// TIA Portal project "ServoPulseHariciPozisyonlama" (V17)

(* hardware
DEVICE "S7-1200 station_1"  S7-1200 Station
   slot 0: "Rack_0"  S7-1200 Rack  Rack  V1.0
   slot 1: "PLC_1"  CPU 1214C DC/DC/DC  6ES7 214-1AG40-0XB0  V4.5
DEVICE "PC-System_1"  SIMATIC PC station
   slot 0: "SIMATIC PC station"  Rail  SIMATIC PC-Station  V1.0
      slot 125: "Stationmanager"  Station_Manager  V6.0.4
   slot 1: "HMI_RT_1"  WinCC RT Advanced  6AV2 104-0xxxx-xxxx  17.0.0.0
      slot 33792: "Computer interface"  Host interface
*)

// ===== PLC "PLC_1"  CPU 1214C DC/DC/DC =====

VAR_GLOBAL   // PLC tag table "Default tag table"
   "Axis_1_Pulse" AT %Q0.0 : Bool;
   "Axis_1_Direction" AT %Q0.1 : Bool;
   "Axis_1_DriveEnable" AT %Q0.2 : Bool;
   "Axis_1_LowHwLimitSwitch" AT %I0.0 : Bool;
   "Axis_1_HighHwLimitSwitch" AT %I0.1 : Bool;
   "SERVO ON/OFF-MC POWER" AT %M0.0 : Bool;
   "Tag_1" AT %M100.0 : Bool;
   "Tag_2" AT %M100.1 : Bool;
   "Tag_3" AT %M100.2 : Bool;
   "Tag_4" AT %MD120 : DWord;
   "Tag_5" AT %MD130 : DWord;
   "Tag_6" AT %MW120 : Word;
   "Tag_7" AT %MW130 : Word;
   "MANUEL İLERİ" AT %M0.1 : Bool;
   "MANUEL GERİ" AT %M0.2 : Bool;
   "MANUEL HIZ DEĞERİ" AT %MD50 : Real;
   "BAŞLANGIÇ NOKTASINA GİT ATA-HOME" AT %M0.3 : Bool;
   "HOME POZİSYON DEĞERİ" AT %MD60 : Real;
   "Tag_10" AT %MB1000 : Byte;
   "HOME MOD DEĞERLERİ" AT %MW1000 : Int;
   "Axis_1_Homing switch" AT %I0.7 : Bool;
   "İSTENEN HEDEFE GİT-ABSOLUTE" AT %M0.4 : Bool;
   "İSTENEN HEDEF-ABSOLUTE" AT %MD100 : Real;
   "HEDEFE GİTME HIZI-ABSOLUTE" AT %MD104 : Real;
   "İSTENEN MESAFE KADAR GİT-RELATİVE" AT %M0.5 : Bool;
   "MESAFE-RELATİVE" AT %MD200 : Real;
   "RELATİVE-HIZ" AT %MD204 : Real;
   "HATA RESET" AT %M0.6 : Bool;
   "RAMPALI DUR-HALT" AT %M0.7 : Bool;
   "MOVE VELOCİTY HIZ ATA" AT %M1.0 : Bool;
   "MOVEVELOCİTY-CURRENT" AT %M1.2 : Bool;
   "PARAMETRE DEĞİŞTİR CHANGEDYNAMİC" AT %M1.3 : Bool;
   "KALKIŞ PARAMETRESİ CHANGE DYNAMİC" AT %M1.4 : Bool;
   "DURMA RAMPASI-CHANGE DYNAMİC" AT %M1.5 : Bool;
   "ACİL STOP DEĞİŞTİR- CHANGE" AT %M1.6 : Bool;
   "YUMUŞATMA ZAMANI DEĞİŞTİR" AT %M1.7 : Bool;
   "HW LİMİT SWİTCH AKTİF" AT %M15.4 : Bool;
   "HW LİMİT SWİTCH PASİF" AT %M15.5 : Bool;
   "SW LİMİT SWİTCH AKTİF" AT %M15.6 : Bool;
   "SW LİMİT SWİTCH PASİF" AT %M15.7 : Bool;
   "VELOCİTY HIZ" AT %M500.0 : Bool;
   "Tag_8" AT %MD500 : Real;
END_VAR

DATA_BLOCK "SERVO MOTOR KONTROLU"   // DB1, Motion_DB
{ S7_Optimized_Access := 'TRUE' }
AUTHOR : SIMATIC
FAMILY : BasicMC
NAME : TO_PosAx
VERSION : 8.0
// stored: InstanceOfName TO_PositioningAxis
"TO_PositioningAxis"
BEGIN
   // Axis.HomingReferencePointSwitch_AddressCU = %I0.7
   // Axis.PositionLimitsMax_AddressCU = %I0.1
   // Axis.PositionLimitsMin_AddressCU = %I0.0
   // Axis.EnableOutput_AddressCU = %Q0.2
   // Axis.DirectionOutputEnabledCU = TRUE
   // Axis.OnlinePtoModeCU = 16#0000_0002
   // Axis.SelectedChannel2EnumCU = %Q0.1
   // Axis.SelectedChannel1EnumCU = %Q0.0
   // Pulse.MinDeltaDeltaFrequencyCU = 0.004
   // Pulse.MaxDeltaDeltaFrequencyCU = 1.0E+10
   // Pulse.MinDeltaFrequencyCU = 0.005
   // Pulse.MaxDeltaFrequencyCU = 9.5E+9
   // Pulse.MinFrequencyCU = 1.0
   // Pulse.MaxFrequencyCU = 100000.0
   // Pulse.OutputSourceCU = 16#0000_0000
   // Axis.SelectPTO = 0
   // Axis.LengthUnitNormalized.Distance = 1013
   // Axis.Encoder.SelectedHscIndexCU = -1
END_DATA_BLOCK

ORGANIZATION_BLOCK "Main"   // OB1, LAD, ProgramCycle
TITLE = "Main Program Sweep (Cycle)"
{ S7_Optimized_Access := 'TRUE' }
VERSION : 0.1
   VAR_INPUT
      Initial_Call : Bool;   // Initial call of this OB
      Remanence : Bool;   // =True, if remanent data are available
   END_VAR
BEGIN

REGION Network 1
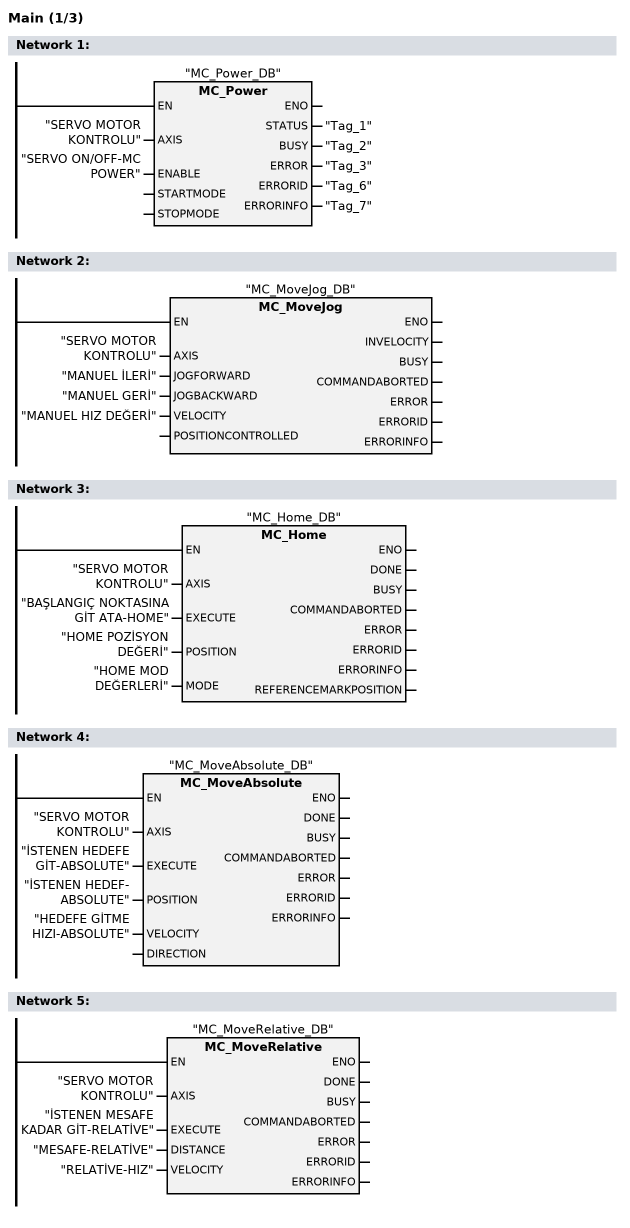
   "MC_Power_DB"(Axis := "SERVO MOTOR KONTROLU",   // MC_Power
                 Enable := "SERVO ON/OFF-MC POWER",
                 Status => "Tag_1",
                 Busy => "Tag_2",
                 Error => "Tag_3",
                 ErrorID => "Tag_6",
                 ErrorInfo => "Tag_7");
END_REGION

REGION Network 2
   "MC_MoveJog_DB"(Axis := "SERVO MOTOR KONTROLU",   // MC_MoveJog
                   JogForward := "MANUEL İLERİ",
                   JogBackward := "MANUEL GERİ",
                   Velocity := "MANUEL HIZ DEĞERİ");
END_REGION

REGION Network 3
   "MC_Home_DB"(Axis := "SERVO MOTOR KONTROLU",   // MC_Home
                Execute := "BAŞLANGIÇ NOKTASINA GİT ATA-HOME",
                Position := "HOME POZİSYON DEĞERİ",
                Mode := "HOME MOD DEĞERLERİ");
END_REGION

REGION Network 4
   "MC_MoveAbsolute_DB"(Axis := "SERVO MOTOR KONTROLU",   // MC_MoveAbsolute
                        Execute := "İSTENEN HEDEFE GİT-ABSOLUTE",
                        Position := "İSTENEN HEDEF-ABSOLUTE",
                        Velocity := "HEDEFE GİTME HIZI-ABSOLUTE");
END_REGION

REGION Network 5
   "MC_MoveRelative_DB"(Axis := "SERVO MOTOR KONTROLU",   // MC_MoveRelative
                        Execute := "İSTENEN MESAFE KADAR GİT-RELATİVE",
                        Distance := "MESAFE-RELATİVE",
                        Velocity := "RELATİVE-HIZ");
END_REGION

REGION Network 6
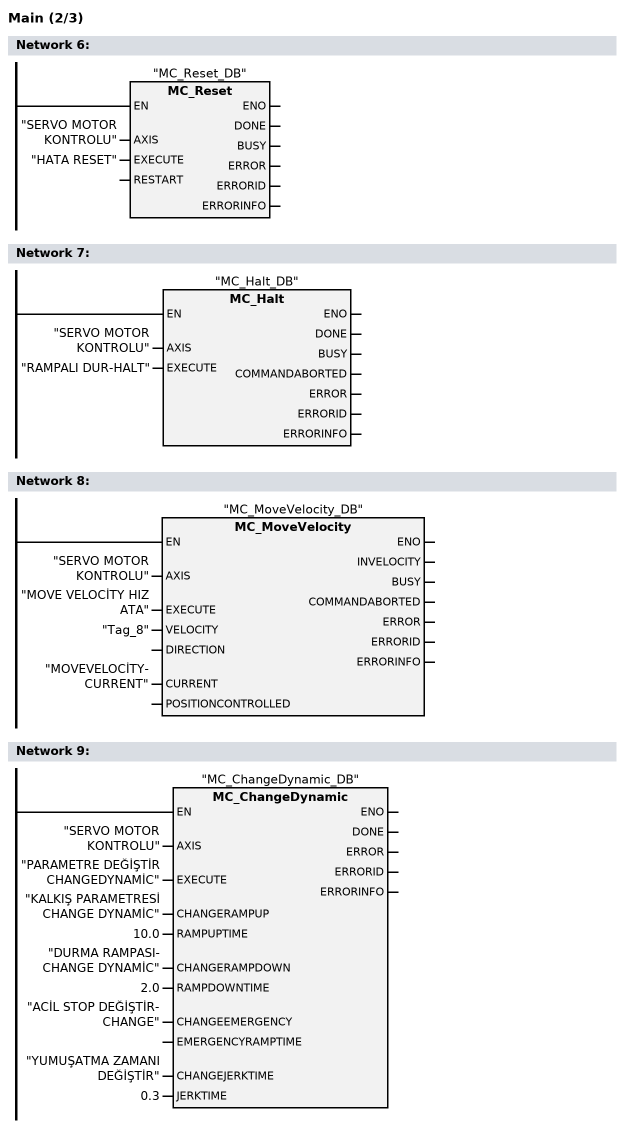
   "MC_Reset_DB"(Axis := "SERVO MOTOR KONTROLU", Execute := "HATA RESET");   // MC_Reset
END_REGION

REGION Network 7
   "MC_Halt_DB"(Axis := "SERVO MOTOR KONTROLU", Execute := "RAMPALI DUR-HALT");   // MC_Halt
END_REGION

REGION Network 8
   "MC_MoveVelocity_DB"(Axis := "SERVO MOTOR KONTROLU",   // MC_MoveVelocity
                        Execute := "MOVE VELOCİTY HIZ ATA",
                        Velocity := "Tag_8",
                        Current := "MOVEVELOCİTY-CURRENT");
END_REGION

REGION Network 9
   "MC_ChangeDynamic_DB"(Axis := "SERVO MOTOR KONTROLU",   // MC_ChangeDynamic
                         Execute := "PARAMETRE DEĞİŞTİR CHANGEDYNAMİC",
                         ChangeRampUp := "KALKIŞ PARAMETRESİ CHANGE DYNAMİC",
                         RampUpTime := 10.0,
                         ChangeRampDown := "DURMA RAMPASI-CHANGE DYNAMİC",
                         RampDownTime := 2.0,
                         ChangeEmergency := "ACİL STOP DEĞİŞTİR- CHANGE",
                         ChangeJerkTime := "YUMUŞATMA ZAMANI DEĞİŞTİR",
                         JerkTime := 0.3);
END_REGION

REGION Network 10
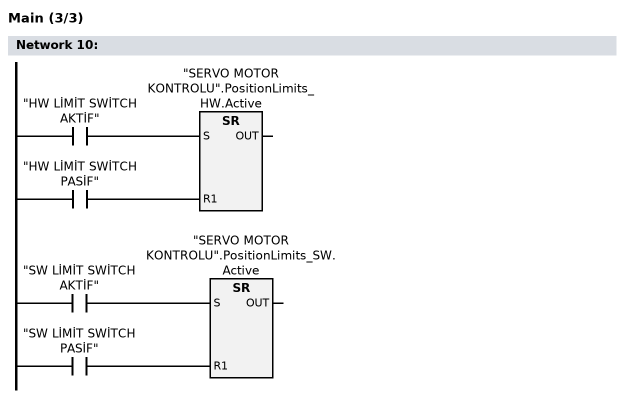
   RUNG wire#powerrail
      Contact( "HW LİMİT SWİTCH AKTİF" )
      S_SR(operand := "SERVO MOTOR KONTROLU".PositionLimits_HW.Active, r1 := wire#w1)
   END_RUNG
   RUNG wire#powerrail
      Contact( "HW LİMİT SWİTCH PASİF" )
   END_RUNG wire#w1
   RUNG wire#powerrail
      Contact( "SW LİMİT SWİTCH AKTİF" )
      S_SR(operand := "SERVO MOTOR KONTROLU".PositionLimits_SW.Active, r1 := wire#w2)
   END_RUNG
   RUNG wire#powerrail
      Contact( "SW LİMİT SWİTCH PASİF" )
   END_RUNG wire#w2
   // the same network as SCL:
   IF "HW LİMİT SWİTCH AKTİF" THEN
       "SERVO MOTOR KONTROLU".PositionLimits_HW.Active := TRUE;   // SR flip-flop
   END_IF;
   IF "HW LİMİT SWİTCH PASİF" THEN "SERVO MOTOR KONTROLU".PositionLimits_HW.Active := FALSE; END_IF;
   IF "SW LİMİT SWİTCH AKTİF" THEN
       "SERVO MOTOR KONTROLU".PositionLimits_SW.Active := TRUE;   // SR flip-flop
   END_IF;
   IF "SW LİMİT SWİTCH PASİF" THEN "SERVO MOTOR KONTROLU".PositionLimits_SW.Active := FALSE; END_IF;
END_REGION
END_ORGANIZATION_BLOCK

(* ===== HMI "HMI_RT_1" =====
system functions are stored by id; their names below are inferred from use
connection "HMI_Connection_1": ETHERNET, S7_1200_OMS

HMI tags "Default tag table"
   "SERVO ON/OFF-MC POWER" : Bool = PLC "SERVO ON/OFF-MC POWER" AT %M0.0, 1 s
   "MANUEL İLERİ" : Bool = PLC "MANUEL İLERİ" AT %M0.1, 1 s
   "MANUEL GERİ" : Bool = PLC "MANUEL GERİ" AT %M0.2, 1 s
   "MANUEL HIZ DEĞERİ" : Real = PLC "MANUEL HIZ DEĞERİ" AT %MD50, 1 s
   "BAŞLANGIÇ NOKTASINA GİT ATA-HOME" : Bool = PLC "BAŞLANGIÇ NOKTASINA GİT ATA-HOME" AT %M0.3, 1 s
   "HOME POZİSYON DEĞERİ" : Real = PLC "HOME POZİSYON DEĞERİ" AT %MD60, 1 s
   "HOME MOD DEĞERLERİ" : Int = PLC "HOME MOD DEĞERLERİ" AT %MW1000, 1 s
   "İSTENEN HEDEFE GİT-ABSOLUTE" : Bool = PLC "İSTENEN HEDEFE GİT-ABSOLUTE" AT %M0.4, 1 s
   "İSTENEN HEDEF-ABSOLUTE" : Real = PLC "İSTENEN HEDEF-ABSOLUTE" AT %MD100, 1 s
   "HEDEFE GİTME HIZI-ABSOLUTE" : Real = PLC "HEDEFE GİTME HIZI-ABSOLUTE" AT %MD104, 1 s
   "İSTENEN MESAFE KADAR GİT-RELATİVE" : Bool = PLC "İSTENEN MESAFE KADAR GİT-RELATİVE" AT %M0.5, 1 s
   "MESAFE-RELATİVE" : Real = PLC "MESAFE-RELATİVE" AT %MD200, 1 s
   "RELATİVE-HIZ" : Real = PLC "RELATİVE-HIZ" AT %MD204, 1 s
   "HATA RESET" : Bool = PLC "HATA RESET" AT %M0.6, 1 s
   "RAMPALI DUR-HALT" : Bool = PLC "RAMPALI DUR-HALT" AT %M0.7, 1 s
   "MOVE VELOCİTY HIZ ATA" : Bool = PLC "MOVE VELOCİTY HIZ ATA" AT %M1.0, 1 s
   "VELOCİTY HIZ" : Bool = PLC "VELOCİTY HIZ" AT %M500.0, 1 s
   "Tag_8" : Real = PLC Tag_8 AT %MD500, 1 s
   "PARAMETRE DEĞİŞTİR CHANGEDYNAMİC" : Bool = PLC "PARAMETRE DEĞİŞTİR CHANGEDYNAMİC" AT %M1.3, 1 s
   "KALKIŞ PARAMETRESİ CHANGE DYNAMİC" : Bool = PLC "KALKIŞ PARAMETRESİ CHANGE DYNAMİC" AT %M1.4, 1 s
   "DURMA RAMPASI-CHANGE DYNAMİC" : Bool = PLC "DURMA RAMPASI-CHANGE DYNAMİC" AT %M1.5, 1 s
   "ACİL STOP DEĞİŞTİR- CHANGE" : Bool = PLC "ACİL STOP DEĞİŞTİR- CHANGE" AT %M1.6, 1 s
   "YUMUŞATMA ZAMANI DEĞİŞTİR" : Bool = PLC "YUMUŞATMA ZAMANI DEĞİŞTİR" AT %M1.7, 1 s

screen "Screen_1" 1920x1080
   TextField "Text field_1" at 71,22 size 95x22; Text 'MC_POWER'
   Button "Button_1" at 33,56 size 172x32; TextOff 'SERVO AKTİF/PASİF'
      on Click: InvertBit("SERVO ON/OFF-MC POWER")
   TextField "Text field_2" at 283,22 size 84x22; Text 'MOVE JOG'
   Button "Button_2" at 261,56 size 137x32; TextOff 'MANUEL İLERİ'
      on Click: InvertBit("MANUEL İLERİ")
   Button "Button_3" at 261,103 size 137x32; TextOff 'MANUEL GERİ'
      on Click: InvertBit("MANUEL GERİ")
   IOField "I/O field_1" at 302,150 size 96x32; FormatPattern 999999
      ProcessValue <- "MANUEL HIZ DEĞERİ"
   TextField "Text field_3" at 230,155 size 72x22; Text 'JOG HIZ:'
   TextField "Text field_4" at 510,22 size 84x22; Text 'MOVE JOG'
   Button "Button_4" at 445,55 size 228x32; TextOff 'BAŞLANGIÇ NOKTASINA GİT'
      on Click: InvertBit("BAŞLANGIÇ NOKTASINA GİT ATA-HOME")
   IOField "I/O field_2" at 594,103 size 96x32; FormatPattern s999999999.999
      ProcessValue <- "HOME POZİSYON DEĞERİ"
   TextField "Text field_5" at 438,109 size 155x22; Text 'POZİSYON DEĞERİ:'
   TextField "Text field_6" at 438,150 size 117x22; Text 'MODE DEĞERİ:'
   IOField "I/O field_3" at 594,145 size 96x32; FormatPattern s99999
      ProcessValue <- "HOME MOD DEĞERLERİ"
   TextField "Text field_7" at 764,22 size 133x22; Text 'MOVE ABSOLUTE'
   Button "Button_5" at 722,56 size 228x32; TextOff 'BAŞLANGIÇ NOKTASINA GİT'
      on Click: InvertBit("İSTENEN HEDEFE GİT-ABSOLUTE")
   TextField "Text field_8" at 722,109 size 155x22; Text 'POZİSYON DEĞERİ:'
   IOField "I/O field_4" at 880,103 size 96x32; FormatPattern s999999999.999
      ProcessValue <- "İSTENEN HEDEF-ABSOLUTE"
   IOField "I/O field_5" at 880,150 size 96x32; FormatPattern s999999999.999
      ProcessValue <- "HEDEFE GİTME HIZI-ABSOLUTE"
   TextField "Text field_9" at 718,155 size 159x22; Text 'HEDEFE GİTME HIZI:'
   TextField "Text field_10" at 1083,22 size 127x22; Text 'MOVE RELATİVE'
   Button "Button_6" at 1032,56 size 228x32; TextOff 'İSTENEN MESAFE KADAR GİT'
      on Click: InvertBit("İSTENEN MESAFE KADAR GİT-RELATİVE")
   TextField "Text field_11" at 1032,109 size 155x22; Text 'POZİSYON DEĞERİ:'
   TextField "Text field_12" at 1028,155 size 37x22; Text 'HIZ:'
   IOField "I/O field_6" at 1193,103 size 96x32; FormatPattern s999999999.999
      ProcessValue <- "MESAFE-RELATİVE"
   IOField "I/O field_7" at 1193,150 size 96x32; FormatPattern s999999999.999
      ProcessValue <- "RELATİVE-HIZ"
   TextField "Text field_13" at 1380,22 size 53x22; Text 'RESET'
   Button "Button_7" at 1363,55 size 94x32; TextOff 'RESET'
      on Click: InvertBit("HATA RESET")
   TextField "Text field_14" at 71,275 size 95x22; Text 'MC_POWER'
   Button "Button_8" at 47,308 size 144x32; TextOff 'RAMPALI DUR'
      on Click: InvertBit("RAMPALI DUR-HALT")
   TextField "Text field_15" at 343,275 size 130x22; Text 'MOVE VELOCİTY'
   Button "Button_9" at 338,308 size 144x32; TextOff 'HIZ ATA'
      on Click: InvertBit("MOVE VELOCİTY HIZ ATA")
   TextField "Text field_16" at 276,362 size 166x22; Text 'ATANAN HIZ DEĞERİ:'
   IOField "I/O field_8" at 446,358 size 96x32; FormatPattern s999999999.999
      ProcessValue <- "Tag_8"
   TextField "Text field_17" at 629,275 size 130x22; Text 'MOVE VELOCİTY'
   Button "Button_10" at 629,308 size 187x32; TextOff 'PARAMETRE DEĞİŞTİR'
      on Click: InvertBit("PARAMETRE DEĞİŞTİR CHANGEDYNAMİC")
   Button "Button_11" at 629,358 size 147x32; TextOff 'KALKIŞ RAMPASI'
      on Click: InvertBit("KALKIŞ PARAMETRESİ CHANGE DYNAMİC")
   Button "Button_12" at 629,408 size 148x32; TextOff 'DURMA RAMPASI'
      on Click: InvertBit("DURMA RAMPASI-CHANGE DYNAMİC")
   Button "Button_13" at 629,458 size 147x32; TextOff 'ACİL DURUM'
      on Click: InvertBit("ACİL STOP DEĞİŞTİR- CHANGE")
   Button "Button_14" at 629,509 size 147x32; TextOff 'YUMUŞATMA'
      on Click: InvertBit("YUMUŞATMA ZAMANI DEĞİŞTİR")
*)